TYPE T_EVENT_CHAR_INDICATOR : STRING(1); END_TYPE

(* stored: Version 1.1.0.1, ProductVersion 3.1.4026.18
   DUT T_EVENT_CHAR_INDICATOR: Id {f4357b37-f183-481f-944c-e42494fc52bf} *)
